   1:  PR[91,1] = PR[90,1] + 27.629;
   1:  PR[91,2] = PR[90,2] + -0.292;
   1:L PR[91] R[100]mm/sec CNT100;
   1:  PR[91,1] = PR[90,1] + 27.566;
   1:  PR[91,2] = PR[90,2] + 0.307;
   1:L PR[91] R[100]mm/sec CNT100;
   1:  PR[91,1] = PR[90,1] + 26.727;
   1:  PR[91,2] = PR[90,2] + 6.678;
   1:L PR[91] R[100]mm/sec CNT100;
   1:  PR[91,1] = PR[90,1] + 26.554;
   1:  PR[91,2] = PR[90,2] + 7.224;
   1:L PR[91] R[100]mm/sec CNT100;
   1:  PR[91,1] = PR[90,1] + 24.093;
   1:  PR[91,2] = PR[90,2] + 13.165;
   1:L PR[91] R[100]mm/sec CNT100;
   1:  PR[91,1] = PR[90,1] + 23.811;
   1:  PR[91,2] = PR[90,2] + 13.670;
   1:L PR[91] R[100]mm/sec CNT100;
   1:  PR[91,1] = PR[90,1] + 19.892;
   1:  PR[91,2] = PR[90,2] + 18.778;
   1:L PR[91] R[100]mm/sec CNT100;
   1:  PR[91,1] = PR[90,1] + 19.473;
   1:  PR[91,2] = PR[90,2] + 19.255;
   1:L PR[91] R[100]mm/sec CNT100;
   1:  PR[91,1] = PR[90,1] + 14.366;
   1:  PR[91,2] = PR[90,2] + 23.173;
   1:L PR[91] R[100]mm/sec CNT100;
   1:  PR[91,1] = PR[90,1] + 13.778;
   1:  PR[91,2] = PR[90,2] + 23.590;
   1:L PR[91] R[100]mm/sec CNT100;
   1:  PR[91,1] = PR[90,1] + 7.843;
   1:  PR[91,2] = PR[90,2] + 26.048;
   1:L PR[91] R[100]mm/sec CNT100;
   1:  PR[91,1] = PR[90,1] + 7.172;
   1:  PR[91,2] = PR[90,2] + 26.308;
   1:L PR[91] R[100]mm/sec CNT100;
   1:  PR[91,1] = PR[90,1] + 0.073;
   1:  PR[91,2] = PR[90,2] + 27.236;
   1:L PR[91] R[100]mm/sec CNT100;
   1:  PR[91] = PR[90];
   1:  PR[91,1] = PR[90,1] + -7.043;
   1:  PR[91,2] = PR[90,2] + 26.299;
   1:  PR[91,3] = PR[90,3] + 80.215;
   1:L PR[91] R[100]mm/sec CNT100;
   1:  PR[91,1] = PR[90,1] + -13.678;
   1:  PR[91,2] = PR[90,2] + 23.555;
   1:L PR[91] R[100]mm/sec CNT100;
   1:  PR[91,1] = PR[90,1] + -19.380;
   1:  PR[91,2] = PR[90,2] + 19.187;
   1:L PR[91] R[100]mm/sec CNT100;
   1:  PR[91,1] = PR[90,1] + -23.783;
   1:  PR[91,2] = PR[90,2] + 13.463;
   1:L PR[91] R[100]mm/sec CNT100;
   1:  PR[91,1] = PR[90,1] + -26.536;
   1:  PR[91,2] = PR[90,2] + 6.793;
   1:L PR[91] R[100]mm/sec CNT100;
   1:  PR[91,1] = PR[90,1] + -27.469;
   1:  PR[91,2] = PR[90,2] + -0.312;
   1:L PR[91] R[100]mm/sec CNT100;
   1:  PR[91,1] = PR[90,1] + -26.533;
   1:  PR[91,2] = PR[90,2] + -7.451;
   1:L PR[91] R[100]mm/sec CNT100;
   1:  PR[91,1] = PR[90,1] + -23.785;
   1:  PR[91,2] = PR[90,2] + -14.085;
   1:L PR[91] R[100]mm/sec CNT100;
   1:  PR[91,1] = PR[90,1] + -19.416;
   1:  PR[91,2] = PR[90,2] + -19.779;
   1:L PR[91] R[100]mm/sec CNT100;
   1:  PR[91,1] = PR[90,1] + -19.389;
   1:  PR[91,2] = PR[90,2] + -19.806;
   1:L PR[91] R[100]mm/sec CNT100;
   1:  PR[91,1] = PR[90,1] + -13.673;
   1:  PR[91,2] = PR[90,2] + -24.181;
   1:L PR[91] R[100]mm/sec CNT100;
   1:  PR[91,1] = PR[90,1] + -7.041;
   1:  PR[91,2] = PR[90,2] + -26.923;
   1:L PR[91] R[100]mm/sec CNT100;
   1:  PR[91,1] = PR[90,1] + 0.101;
   1:  PR[91,2] = PR[90,2] + -27.862;
   1:L PR[91] R[100]mm/sec CNT100;
   1:  PR[91,1] = PR[90,1] + 7.204;
   1:  PR[91,2] = PR[90,2] + -26.922;
   1:L PR[91] R[100]mm/sec CNT100;
   1:  PR[91,1] = PR[90,1] + 13.835;
   1:  PR[91,2] = PR[90,2] + -24.178;
   1:L PR[91] R[100]mm/sec CNT100;
   1:  PR[91,1] = PR[90,1] + 19.567;
   1:  PR[91,2] = PR[90,2] + -19.788;
   1:L PR[91] R[100]mm/sec CNT100;
   1:  PR[91,1] = PR[90,1] + 23.940;
   1:  PR[91,2] = PR[90,2] + -14.088;
   1:L PR[91] R[100]mm/sec CNT100;
   1:  PR[91,1] = PR[90,1] + 26.688;
   1:  PR[91,2] = PR[90,2] + -7.452;
   1:L PR[91] R[100]mm/sec CNT100;
   1:  PR[91,1] = PR[90,1] + 27.626;
   1:  PR[91,2] = PR[90,2] + -0.312;
   1:L PR[91] R[100]mm/sec CNT100;
   1:  PR[91,1] = PR[90,1] + 26.689;
   1:  PR[91,2] = PR[90,2] + 6.827;
   1:L PR[91] R[100]mm/sec CNT100;
   1:  PR[91,1] = PR[90,1] + 23.942;
   1:  PR[91,2] = PR[90,2] + 13.461;
   1:L PR[91] R[100]mm/sec CNT100;
   1:  PR[91,1] = PR[90,1] + 19.566;
   1:  PR[91,2] = PR[90,2] + 19.165;
   1:L PR[91] R[100]mm/sec CNT100;
   1:  PR[91,1] = PR[90,1] + 13.834;
   1:  PR[91,2] = PR[90,2] + 23.555;
   1:L PR[91] R[100]mm/sec CNT100;
   1:  PR[91,1] = PR[90,1] + 7.200;
   1:  PR[91,2] = PR[90,2] + 26.299;
   1:L PR[91] R[100]mm/sec CNT100;
   1:  PR[91,1] = PR[90,1] + 0.078;
   1:  PR[91,2] = PR[90,2] + 27.237;
   1:L PR[91] R[100]mm/sec CNT100;
   1:  PR[91,1] = PR[90,1] + -7.043;
   1:  PR[91,2] = PR[90,2] + 26.299;
   1:L PR[91] R[100]mm/sec CNT100;
   1:  PR[91,1] = PR[90,1] + -13.678;
   1:  PR[91,2] = PR[90,2] + 23.555;
   1:L PR[91] R[100]mm/sec CNT100;
   1:  PR[91,1] = PR[90,1] + -19.380;
   1:  PR[91,2] = PR[90,2] + 19.187;
   1:L PR[91] R[100]mm/sec CNT100;
   1:  PR[91,1] = PR[90,1] + -23.783;
   1:  PR[91,2] = PR[90,2] + 13.463;
   1:L PR[91] R[100]mm/sec CNT100;
   1:  PR[91,1] = PR[90,1] + -26.536;
   1:  PR[91,2] = PR[90,2] + 6.793;
   1:L PR[91] R[100]mm/sec CNT100;
   1:  PR[91,1] = PR[90,1] + -27.469;
   1:  PR[91,2] = PR[90,2] + -0.312;
   1:L PR[91] R[100]mm/sec CNT100;
   1:  PR[91,1] = PR[90,1] + -26.533;
   1:  PR[91,2] = PR[90,2] + -7.451;
   1:L PR[91] R[100]mm/sec CNT100;
   1:  PR[91,1] = PR[90,1] + -23.785;
   1:  PR[91,2] = PR[90,2] + -14.085;
   1:L PR[91] R[100]mm/sec CNT100;
   1:  PR[91,1] = PR[90,1] + -19.416;
   1:  PR[91,2] = PR[90,2] + -19.779;
   1:L PR[91] R[100]mm/sec CNT100;
   1:  PR[91,1] = PR[90,1] + -19.389;
   1:  PR[91,2] = PR[90,2] + -19.806;
   1:L PR[91] R[100]mm/sec CNT100;
   1:  PR[91,1] = PR[90,1] + -13.673;
   1:  PR[91,2] = PR[90,2] + -24.181;
   1:L PR[91] R[100]mm/sec CNT100;
   1:  PR[91,1] = PR[90,1] + -7.041;
   1:  PR[91,2] = PR[90,2] + -26.923;
   1:L PR[91] R[100]mm/sec CNT100;
   1:  PR[91,1] = PR[90,1] + 0.101;
   1:  PR[91,2] = PR[90,2] + -27.862;
   1:L PR[91] R[100]mm/sec CNT100;
   1:  PR[91,1] = PR[90,1] + 7.204;
   1:  PR[91,2] = PR[90,2] + -26.922;
   1:L PR[91] R[100]mm/sec CNT100;
   1:  PR[91,1] = PR[90,1] + 13.835;
   1:  PR[91,2] = PR[90,2] + -24.178;
   1:L PR[91] R[100]mm/sec CNT100;
   1:  PR[91,1] = PR[90,1] + 19.567;
   1:  PR[91,2] = PR[90,2] + -19.788;
   1:L PR[91] R[100]mm/sec CNT100;
   1:  PR[91,1] = PR[90,1] + 23.940;
   1:  PR[91,2] = PR[90,2] + -14.088;
   1:L PR[91] R[100]mm/sec CNT100;
   1:  PR[91,1] = PR[90,1] + 26.688;
   1:  PR[91,2] = PR[90,2] + -7.452;
   1:L PR[91] R[100]mm/sec CNT100;
   1:  PR[91,1] = PR[90,1] + 27.626;
   1:  PR[91,2] = PR[90,2] + -0.312;
   1:L PR[91] R[100]mm/sec CNT100;
   1:  PR[91,1] = PR[90,1] + 26.689;
   1:  PR[91,2] = PR[90,2] + 6.827;
   1:L PR[91] R[100]mm/sec CNT100;
   1:  PR[91,1] = PR[90,1] + 23.942;
   1:  PR[91,2] = PR[90,2] + 13.461;
   1:L PR[91] R[100]mm/sec CNT100;
   1:  PR[91,1] = PR[90,1] + 19.566;
   1:  PR[91,2] = PR[90,2] + 19.165;
   1:L PR[91] R[100]mm/sec CNT100;
   1:  PR[91,1] = PR[90,1] + 13.834;
   1:  PR[91,2] = PR[90,2] + 23.555;
   1:L PR[91] R[100]mm/sec CNT100;
   1:  PR[91,1] = PR[90,1] + 7.200;
   1:  PR[91,2] = PR[90,2] + 26.299;
   1:L PR[91] R[100]mm/sec CNT100;
   1:  PR[91,1] = PR[90,1] + 0.078;
   1:  PR[91,2] = PR[90,2] + 27.237;
   1:L PR[91] R[100]mm/sec CNT100 TB   .50sec,CALL END_PUD;
   1:  DO[117:Laser Start]=OFF;
   1:  PR[92] = PR[91];
   1:  PR[92,3] = PR[92,3] + 50;
   1:J PR[92] 10% FINE;
   1:  WAIT   5.00(sec);
   1:  DO[119:Gas]=OFF;
   1:  CALL HOME_ALL;
/POS
/END
